   cmAnodeMainPnP2AxisZ.commandConfiguration.posRelative.direction := 0;
   cmAnodeMainPnP2AxisZ.commandConfiguration.posAbsolute.position := 3.0;
   cmAnodeMainPnP2AxisZ.commandConfiguration.posAbsolute.velocity := 30.0;
   cmAnodeMainPnP2AxisZ.commandConfiguration.posAbsolute.acceleration := 30.0;
   cmAnodeMainPnP2AxisZ.commandConfiguration.posAbsolute.deceleration := 30.0;
   cmAnodeMainPnP2AxisZ.commandConfiguration.posAbsolute.jerk := -1.0;
   cmAnodeMainPnP2AxisZ.commandConfiguration.posAbsolute.direction := 1;
   cmAnodeMainPnP2AxisZ.commandConfiguration.posAbsolute.positionChangeOnTheFly := FALSE;
   cmAnodeMainPnP2AxisZ.commandConfiguration.posAbsolute.velocityChangeOnTheFly := FALSE;
   cmAnodeMainPnP2AxisZ.commandConfiguration.posSuperimposed.distance := 0.0;
   cmAnodeMainPnP2AxisZ.commandConfiguration.posSuperimposed.velocityDiff := -1.0;
   cmAnodeMainPnP2AxisZ.commandConfiguration.posSuperimposed.acceleration := -1.0;
   cmAnodeMainPnP2AxisZ.commandConfiguration.posSuperimposed.deceleration := -1.0;
   cmAnodeMainPnP2AxisZ.commandConfiguration.posSuperimposed.jerk := -1.0;
   cmAnodeMainPnP2AxisZ.commandConfiguration.posSuperimposed.direction := 0;
   cmAnodeMainPnP2AxisZ.commandConfiguration.haltSuperimposed.deceleration := -1.0;
   cmAnodeMainPnP2AxisZ.commandConfiguration.haltSuperimposed.jerk := -1.0;
   cmAnodeMainPnP2AxisZ.commandConfiguration.haltSuperimposed.abortAcceleration := FALSE;
   cmAnodeMainPnP2AxisZ.commandConfiguration.gearInRelative.ratioNumerator := 1;
   cmAnodeMainPnP2AxisZ.commandConfiguration.gearInRelative.ratioDenominator := 1;
   cmAnodeMainPnP2AxisZ.commandConfiguration.gearInRelative.acceleration := -1.0;
   cmAnodeMainPnP2AxisZ.commandConfiguration.gearInRelative.deceleration := -1.0;
   cmAnodeMainPnP2AxisZ.commandConfiguration.gearInRelative.jerk := -1.0;
   cmAnodeMainPnP2AxisZ.commandConfiguration.gearInRelative.ratioChangeOnTheFly := FALSE;
   cmAnodeMainPnP2AxisZ.commandConfiguration.gearInAbsolute.ratioNumerator := 1;
   cmAnodeMainPnP2AxisZ.commandConfiguration.gearInAbsolute.ratioDenominator := 1;
   cmAnodeMainPnP2AxisZ.commandConfiguration.gearInAbsolute.masterSyncPosition := 0.0;
   cmAnodeMainPnP2AxisZ.commandConfiguration.gearInAbsolute.slaveSyncPosition := 0.0;
   cmAnodeMainPnP2AxisZ.commandConfiguration.gearInAbsolute.syncProfileReference := 1;
   cmAnodeMainPnP2AxisZ.commandConfiguration.gearInAbsolute.masterStartDistance := 0.0;
   cmAnodeMainPnP2AxisZ.commandConfiguration.gearInAbsolute.velocity := -1.0;
   cmAnodeMainPnP2AxisZ.commandConfiguration.gearInAbsolute.acceleration := -1.0;
   cmAnodeMainPnP2AxisZ.commandConfiguration.gearInAbsolute.deceleration := -1.0;
   cmAnodeMainPnP2AxisZ.commandConfiguration.gearInAbsolute.jerk := -1.0;
   cmAnodeMainPnP2AxisZ.commandConfiguration.gearInAbsolute.syncDirection := 1;
   cmAnodeMainPnP2AxisZ.commandConfiguration.gearInAbsolute.ratioChangeOnTheFly := FALSE;
   cmAnodeMainPnP2AxisZ.commandConfiguration.gearInVelocity.continuousUpdate := FALSE;
   cmAnodeMainPnP2AxisZ.commandConfiguration.gearInVelocity.ratioNumerator := 1;
   cmAnodeMainPnP2AxisZ.commandConfiguration.gearInVelocity.ratioDenominator := 1;
   cmAnodeMainPnP2AxisZ.commandConfiguration.gearInVelocity.acceleration := -1.0;
   cmAnodeMainPnP2AxisZ.commandConfiguration.gearInVelocity.deceleration := -1.0;
   cmAnodeMainPnP2AxisZ.commandConfiguration.gearInVelocity.jerk := -1.0;
   cmAnodeMainPnP2AxisZ.commandConfiguration.gearInVelocity.positionControlled := FALSE;
   cmAnodeMainPnP2AxisZ.commandConfiguration.camIn.masterOffset := 0.0;
   cmAnodeMainPnP2AxisZ.commandConfiguration.camIn.slaveOffset := 0.0;
   cmAnodeMainPnP2AxisZ.commandConfiguration.camIn.masterScaling := 1.0;
   cmAnodeMainPnP2AxisZ.commandConfiguration.camIn.slaveScaling := 1.0;
   cmAnodeMainPnP2AxisZ.commandConfiguration.camIn.masterSyncPosition := 0.0;
   cmAnodeMainPnP2AxisZ.commandConfiguration.camIn.syncProfileReference := 1;
   cmAnodeMainPnP2AxisZ.commandConfiguration.camIn.masterStartDistance := 0.0;
   cmAnodeMainPnP2AxisZ.commandConfiguration.camIn.velocity := -1.0;
   cmAnodeMainPnP2AxisZ.commandConfiguration.camIn.acceleration := -1.0;
   cmAnodeMainPnP2AxisZ.commandConfiguration.camIn.deceleration := -1.0;
   cmAnodeMainPnP2AxisZ.commandConfiguration.camIn.jerk := -1.0;
   cmAnodeMainPnP2AxisZ.commandConfiguration.camIn.applicationMode := 0;
   cmAnodeMainPnP2AxisZ.commandConfiguration.camIn.syncDirection := 1;
   cmAnodeMainPnP2AxisZ.commandConfiguration.gearOutCamOut.slavePosition := 0.0;
   cmAnodeMainPnP2AxisZ.commandConfiguration.gearOutCamOut.syncProfileReference := 1;
   cmAnodeMainPnP2AxisZ.commandConfiguration.gearOutCamOut.masterStopDistance := 0.0;
   cmAnodeMainPnP2AxisZ.commandConfiguration.gearOutCamOut.deceleration := -1.0;
   cmAnodeMainPnP2AxisZ.commandConfiguration.gearOutCamOut.jerk := -1.0;
   cmAnodeMainPnP2AxisZ.commandConfiguration.gearOutCamOut.syncOutDirection := 3;
   cmAnodeMainPnP2AxisZ.commandConfiguration.gearOutCamOut.gearOutCamOutMode := -1;
   cmAnodeMainPnP2AxisZ.commandConfiguration.phasing.phaseShift := 0.0;
   cmAnodeMainPnP2AxisZ.commandConfiguration.phasing.velocity := -1.0;
   cmAnodeMainPnP2AxisZ.commandConfiguration.phasing.acceleration := -1.0;
   cmAnodeMainPnP2AxisZ.commandConfiguration.phasing.deceleration := -1.0;
   cmAnodeMainPnP2AxisZ.commandConfiguration.phasing.jerk := -1.0;
   cmAnodeMainPnP2AxisZ.commandConfiguration.phasing.profileReference := 0;
   cmAnodeMainPnP2AxisZ.commandConfiguration.phasing.phasingDistance := 0.0;
   cmAnodeMainPnP2AxisZ.commandConfiguration.phasing.startPosition := 0.0;
   cmAnodeMainPnP2AxisZ.commandConfiguration.phasing.direction := 3;
   cmAnodeMainPnP2AxisZ.commandConfiguration.phasing.phaseAbsolute := TRUE;
   cmAnodeMainPnP2AxisZ.commandConfiguration.phasing.phaseShiftChangeOnTheFly := FALSE;
   cmAnodeMainPnP2AxisZ.commandConfiguration.offset.offset := 0.0;
   cmAnodeMainPnP2AxisZ.commandConfiguration.offset.profileReference := 1;
   cmAnodeMainPnP2AxisZ.commandConfiguration.offset.offsetDistance := 0.0;
   cmAnodeMainPnP2AxisZ.commandConfiguration.offset.startPosition := 0.0;
   cmAnodeMainPnP2AxisZ.commandConfiguration.offset.direction := 3;
   cmAnodeMainPnP2AxisZ.commandConfiguration.offset.offsetAbsolute := TRUE;
   cmAnodeMainPnP2AxisZ.commandConfiguration.offset.offsetChangeOnTheFly := FALSE;
   cmAnodeMainPnP2AxisZ.commands.enableAxis := FALSE;
   cmAnodeMainPnP2AxisZ.commands.resetAxis := FALSE;
   cmAnodeMainPnP2AxisZ.commands.openBrake := FALSE;
   cmAnodeMainPnP2AxisZ.commands.jogForward := FALSE;
   cmAnodeMainPnP2AxisZ.commands.jogBackward := FALSE;
   cmAnodeMainPnP2AxisZ.commands.moveVelocity := FALSE;
   cmAnodeMainPnP2AxisZ.commands.stop := FALSE;
   cmAnodeMainPnP2AxisZ.commands.fastStop := FALSE;
   cmAnodeMainPnP2AxisZ.commands.torqueLimiting := FALSE;
   cmAnodeMainPnP2AxisZ.commands.homing := FALSE;
   cmAnodeMainPnP2AxisZ.commands.posRelative := FALSE;
   cmAnodeMainPnP2AxisZ.commands.posAbsolute := FALSE;
   cmAnodeMainPnP2AxisZ.commands.posSuperimposed := FALSE;
   cmAnodeMainPnP2AxisZ.commands.haltSuperimposed := FALSE;
   cmAnodeMainPnP2AxisZ.commands.selectSetPosition := -1;
   cmAnodeMainPnP2AxisZ.commands.reset := FALSE;
   cmAnodeMainPnP2AxisZ.monitoring.valid := FALSE;
   cmAnodeMainPnP2AxisZ.monitoring.busy := TRUE;
   cmAnodeMainPnP2AxisZ.monitoring.error := TRUE;
   cmAnodeMainPnP2AxisZ.monitoring.status := 16#8600;
   cmAnodeMainPnP2AxisZ.monitoring.subfunctionStatus := 16#8001;
   cmAnodeMainPnP2AxisZ.monitoring.axisEnabled := FALSE;
   cmAnodeMainPnP2AxisZ.monitoring.resetActive := FALSE;
   cmAnodeMainPnP2AxisZ.monitoring.inVelocity := FALSE;
   cmAnodeMainPnP2AxisZ.monitoring.inLimitation := FALSE;
   cmAnodeMainPnP2AxisZ.monitoring.inClamping := FALSE;
   cmAnodeMainPnP2AxisZ.monitoring.startSync := FALSE;
   cmAnodeMainPnP2AxisZ.monitoring.inSync := FALSE;
   cmAnodeMainPnP2AxisZ.monitoring.inSimulation := FALSE;
   cmAnodeMainPnP2AxisZ.monitoring.jogSelected := FALSE;
   cmAnodeMainPnP2AxisZ.monitoring.moveVelocitySelected := FALSE;
   cmAnodeMainPnP2AxisZ.monitoring.stopSelected := FALSE;
   cmAnodeMainPnP2AxisZ.monitoring.fastStopSelected := FALSE;
   cmAnodeMainPnP2AxisZ.monitoring.torqueLimitingSelected := FALSE;
   cmAnodeMainPnP2AxisZ.monitoring.homingSelected := FALSE;
   cmAnodeMainPnP2AxisZ.monitoring.posRelativeSelected := FALSE;
   cmAnodeMainPnP2AxisZ.monitoring.posAbsoluteSelected := FALSE;
   cmAnodeMainPnP2AxisZ.monitoring.posSuperimposedSelected := FALSE;
   cmAnodeMainPnP2AxisZ.monitoring.haltSuperimposedSelected := FALSE;
   cmAnodeMainPnP2AxisZ.monitoring.commandBusy := FALSE;
   cmAnodeMainPnP2AxisZ.monitoring.commandDone := FALSE;
   cmAnodeMainPnP2AxisZ.monitoring.commandAborted := FALSE;
   cmAnodeMainPnP2AxisZ.monitoring.homingCommandBusy := FALSE;
   cmAnodeMainPnP2AxisZ.monitoring.homingCommandDone := FALSE;
   cmAnodeMainPnP2AxisZ.monitoring.homingCommandAborted := FALSE;
   cmAnodeMainPnP2AxisZ.monitoring.superimposedBusy := FALSE;
   cmAnodeMainPnP2AxisZ.monitoring.superimposedDone := FALSE;
   cmAnodeMainPnP2AxisZ.monitoring.superimposedAborted := FALSE;
   cmAnodeMainPnP2AxisZ.monitoring.actualPosition := 3.014;
   cmAnodeMainPnP2AxisZ.monitoring.actualSpeed := -0.00158945719401042;
   cmAnodeMainPnP2AxisZ.monitoring.speedUnit := 1062;
   cmAnodeMainPnP2AxisZ.monitoring.positionUnit := 1013;
   cmAnodeMainPnP2AxisZ.monitoring.axisType := 1;
   cmAnodeMainPnP2AxisZ.monitoring.interlockGeneralOut := TRUE;
   cmAnodeMainPnP2AxisZ.monitoring.interlockJogForwardOut := TRUE;
   cmAnodeMainPnP2AxisZ.monitoring.interlockJogBackwardOut := TRUE;
   cmAnodeAlignTableAxisX.commandConfiguration.generalSettings.stopOnError := TRUE;
   cmAnodeAlignTableAxisX.commandConfiguration.generalSettings.resetWithRestart := FALSE;
   cmAnodeAlignTableAxisX.commandConfiguration.generalSettings.abortWaitingSyncCmd := TRUE;
   cmAnodeAlignTableAxisX.commandConfiguration.power.startMode := 1;
   cmAnodeAlignTableAxisX.commandConfiguration.power.stopMode := 0;
   cmAnodeAlignTableAxisX.commandConfiguration.power.syncMotionSimulation := FALSE;
   cmAnodeAlignTableAxisX.commandConfiguration.power.syncMotionSimulationExtendedMode := -1;
   cmAnodeAlignTableAxisX.commandConfiguration.jog.velocity := 0.0;
   cmAnodeAlignTableAxisX.commandConfiguration.jog.acceleration := -1.0;
   cmAnodeAlignTableAxisX.commandConfiguration.jog.deceleration := -1.0;
   cmAnodeAlignTableAxisX.commandConfiguration.jog.jerk := -1.0;
   cmAnodeAlignTableAxisX.commandConfiguration.jog.positionControlled := TRUE;
   cmAnodeAlignTableAxisX.commandConfiguration.jog.increment := 0.0;
   cmAnodeAlignTableAxisX.commandConfiguration.jog.mode := 0;
   cmAnodeAlignTableAxisX.commandConfiguration.moveVelocity.velocity := 0.0;
   cmAnodeAlignTableAxisX.commandConfiguration.moveVelocity.acceleration := -1.0;
   cmAnodeAlignTableAxisX.commandConfiguration.moveVelocity.deceleration := -1.0;
   cmAnodeAlignTableAxisX.commandConfiguration.moveVelocity.jerk := -1.0;
   cmAnodeAlignTableAxisX.commandConfiguration.moveVelocity.direction := 0;
   cmAnodeAlignTableAxisX.commandConfiguration.moveVelocity.positionControlled := TRUE;
   cmAnodeAlignTableAxisX.commandConfiguration.moveVelocity.velocityChangeOnTheFly := FALSE;
   cmAnodeAlignTableAxisX.commandConfiguration.stop.deceleration := -1.0;
   cmAnodeAlignTableAxisX.commandConfiguration.stop.jerk := -1.0;
   cmAnodeAlignTableAxisX.commandConfiguration.stop.abortAcceleration := FALSE;
   cmAnodeAlignTableAxisX.commandConfiguration.fastStop.deceleration := -1.0;
   cmAnodeAlignTableAxisX.commandConfiguration.fastStop.jerk := -1.0;
   cmAnodeAlignTableAxisX.commandConfiguration.fastStop.abortAcceleration := FALSE;
   cmAnodeAlignTableAxisX.commandConfiguration.fastStop.replaceStopPossible := FALSE;
   cmAnodeAlignTableAxisX.commandConfiguration.torqueLimiting.limit := -1.0;
   cmAnodeAlignTableAxisX.commandConfiguration.torqueLimiting.mode := 0;
   cmAnodeAlignTableAxisX.commandConfiguration.homing.position := 0.0;
   cmAnodeAlignTableAxisX.commandConfiguration.homing.mode := 0;
   cmAnodeAlignTableAxisX.commandConfiguration.homing.sensor := 0;
   cmAnodeAlignTableAxisX.commandConfiguration.homing.extendedMode := -1;
   cmAnodeAlignTableAxisX.commandConfiguration.homing.extendedModeTorqueLimit := 0.0;
   cmAnodeAlignTableAxisX.commandConfiguration.homing.extendedModeTargetPosition := 0.0;
   cmAnodeAlignTableAxisX.commandConfiguration.posRelative.distance := 0.0;
   cmAnodeAlignTableAxisX.commandConfiguration.posRelative.velocity := -1.0;
   cmAnodeAlignTableAxisX.commandConfiguration.posRelative.acceleration := -1.0;
   cmAnodeAlignTableAxisX.commandConfiguration.posRelative.deceleration := -1.0;
   cmAnodeAlignTableAxisX.commandConfiguration.posRelative.jerk := -1.0;
   cmAnodeAlignTableAxisX.commandConfiguration.posRelative.direction := 0;
   cmAnodeAlignTableAxisX.commandConfiguration.posAbsolute.position := 0.0;
   cmAnodeAlignTableAxisX.commandConfiguration.posAbsolute.velocity := -1.0;
   cmAnodeAlignTableAxisX.commandConfiguration.posAbsolute.acceleration := -1.0;
   cmAnodeAlignTableAxisX.commandConfiguration.posAbsolute.deceleration := -1.0;
   cmAnodeAlignTableAxisX.commandConfiguration.posAbsolute.jerk := -1.0;
   cmAnodeAlignTableAxisX.commandConfiguration.posAbsolute.direction := 1;
   cmAnodeAlignTableAxisX.commandConfiguration.posAbsolute.positionChangeOnTheFly := FALSE;
   cmAnodeAlignTableAxisX.commandConfiguration.posAbsolute.velocityChangeOnTheFly := FALSE;
   cmAnodeAlignTableAxisX.commandConfiguration.posSuperimposed.distance := 0.0;
   cmAnodeAlignTableAxisX.commandConfiguration.posSuperimposed.velocityDiff := -1.0;
   cmAnodeAlignTableAxisX.commandConfiguration.posSuperimposed.acceleration := -1.0;
   cmAnodeAlignTableAxisX.commandConfiguration.posSuperimposed.deceleration := -1.0;
   cmAnodeAlignTableAxisX.commandConfiguration.posSuperimposed.jerk := -1.0;
   cmAnodeAlignTableAxisX.commandConfiguration.posSuperimposed.direction := 0;
   cmAnodeAlignTableAxisX.commandConfiguration.haltSuperimposed.deceleration := -1.0;
   cmAnodeAlignTableAxisX.commandConfiguration.haltSuperimposed.jerk := -1.0;
   cmAnodeAlignTableAxisX.commandConfiguration.haltSuperimposed.abortAcceleration := FALSE;
   cmAnodeAlignTableAxisX.commandConfiguration.gearInRelative.ratioNumerator := 1;
   cmAnodeAlignTableAxisX.commandConfiguration.gearInRelative.ratioDenominator := 1;
   cmAnodeAlignTableAxisX.commandConfiguration.gearInRelative.acceleration := -1.0;
   cmAnodeAlignTableAxisX.commandConfiguration.gearInRelative.deceleration := -1.0;
   cmAnodeAlignTableAxisX.commandConfiguration.gearInRelative.jerk := -1.0;
   cmAnodeAlignTableAxisX.commandConfiguration.gearInRelative.ratioChangeOnTheFly := FALSE;
   cmAnodeAlignTableAxisX.commandConfiguration.gearInAbsolute.ratioNumerator := 1;
   cmAnodeAlignTableAxisX.commandConfiguration.gearInAbsolute.ratioDenominator := 1;
   cmAnodeAlignTableAxisX.commandConfiguration.gearInAbsolute.masterSyncPosition := 0.0;
   cmAnodeAlignTableAxisX.commandConfiguration.gearInAbsolute.slaveSyncPosition := 0.0;
   cmAnodeAlignTableAxisX.commandConfiguration.gearInAbsolute.syncProfileReference := 1;
   cmAnodeAlignTableAxisX.commandConfiguration.gearInAbsolute.masterStartDistance := 0.0;
   cmAnodeAlignTableAxisX.commandConfiguration.gearInAbsolute.velocity := -1.0;
   cmAnodeAlignTableAxisX.commandConfiguration.gearInAbsolute.acceleration := -1.0;
   cmAnodeAlignTableAxisX.commandConfiguration.gearInAbsolute.deceleration := -1.0;
   cmAnodeAlignTableAxisX.commandConfiguration.gearInAbsolute.jerk := -1.0;
   cmAnodeAlignTableAxisX.commandConfiguration.gearInAbsolute.syncDirection := 1;
   cmAnodeAlignTableAxisX.commandConfiguration.gearInAbsolute.ratioChangeOnTheFly := FALSE;
   cmAnodeAlignTableAxisX.commandConfiguration.gearInVelocity.continuousUpdate := FALSE;
   cmAnodeAlignTableAxisX.commandConfiguration.gearInVelocity.ratioNumerator := 1;
   cmAnodeAlignTableAxisX.commandConfiguration.gearInVelocity.ratioDenominator := 1;
   cmAnodeAlignTableAxisX.commandConfiguration.gearInVelocity.acceleration := -1.0;
   cmAnodeAlignTableAxisX.commandConfiguration.gearInVelocity.deceleration := -1.0;
   cmAnodeAlignTableAxisX.commandConfiguration.gearInVelocity.jerk := -1.0;
   cmAnodeAlignTableAxisX.commandConfiguration.gearInVelocity.positionControlled := FALSE;
   cmAnodeAlignTableAxisX.commandConfiguration.camIn.masterOffset := 0.0;
   cmAnodeAlignTableAxisX.commandConfiguration.camIn.slaveOffset := 0.0;
   cmAnodeAlignTableAxisX.commandConfiguration.camIn.masterScaling := 1.0;
   cmAnodeAlignTableAxisX.commandConfiguration.camIn.slaveScaling := 1.0;
   cmAnodeAlignTableAxisX.commandConfiguration.camIn.masterSyncPosition := 0.0;
   cmAnodeAlignTableAxisX.commandConfiguration.camIn.syncProfileReference := 1;
   cmAnodeAlignTableAxisX.commandConfiguration.camIn.masterStartDistance := 0.0;
   cmAnodeAlignTableAxisX.commandConfiguration.camIn.velocity := -1.0;
   cmAnodeAlignTableAxisX.commandConfiguration.camIn.acceleration := -1.0;
   cmAnodeAlignTableAxisX.commandConfiguration.camIn.deceleration := -1.0;
   cmAnodeAlignTableAxisX.commandConfiguration.camIn.jerk := -1.0;
   cmAnodeAlignTableAxisX.commandConfiguration.camIn.applicationMode := 0;
   cmAnodeAlignTableAxisX.commandConfiguration.camIn.syncDirection := 1;
   cmAnodeAlignTableAxisX.commandConfiguration.gearOutCamOut.slavePosition := 0.0;
   cmAnodeAlignTableAxisX.commandConfiguration.gearOutCamOut.syncProfileReference := 1;
   cmAnodeAlignTableAxisX.commandConfiguration.gearOutCamOut.masterStopDistance := 0.0;
   cmAnodeAlignTableAxisX.commandConfiguration.gearOutCamOut.deceleration := -1.0;
   cmAnodeAlignTableAxisX.commandConfiguration.gearOutCamOut.jerk := -1.0;
   cmAnodeAlignTableAxisX.commandConfiguration.gearOutCamOut.syncOutDirection := 3;
   cmAnodeAlignTableAxisX.commandConfiguration.gearOutCamOut.gearOutCamOutMode := -1;
   cmAnodeAlignTableAxisX.commandConfiguration.phasing.phaseShift := 0.0;
   cmAnodeAlignTableAxisX.commandConfiguration.phasing.velocity := -1.0;
   cmAnodeAlignTableAxisX.commandConfiguration.phasing.acceleration := -1.0;
   cmAnodeAlignTableAxisX.commandConfiguration.phasing.deceleration := -1.0;
   cmAnodeAlignTableAxisX.commandConfiguration.phasing.jerk := -1.0;
   cmAnodeAlignTableAxisX.commandConfiguration.phasing.profileReference := 0;
   cmAnodeAlignTableAxisX.commandConfiguration.phasing.phasingDistance := 0.0;
   cmAnodeAlignTableAxisX.commandConfiguration.phasing.startPosition := 0.0;
   cmAnodeAlignTableAxisX.commandConfiguration.phasing.direction := 3;
   cmAnodeAlignTableAxisX.commandConfiguration.phasing.phaseAbsolute := TRUE;
   cmAnodeAlignTableAxisX.commandConfiguration.phasing.phaseShiftChangeOnTheFly := FALSE;
   cmAnodeAlignTableAxisX.commandConfiguration.offset.offset := 0.0;
   cmAnodeAlignTableAxisX.commandConfiguration.offset.profileReference := 1;
   cmAnodeAlignTableAxisX.commandConfiguration.offset.offsetDistance := 0.0;
   cmAnodeAlignTableAxisX.commandConfiguration.offset.startPosition := 0.0;
   cmAnodeAlignTableAxisX.commandConfiguration.offset.direction := 3;
   cmAnodeAlignTableAxisX.commandConfiguration.offset.offsetAbsolute := TRUE;
   cmAnodeAlignTableAxisX.commandConfiguration.offset.offsetChangeOnTheFly := FALSE;
   cmAnodeAlignTableAxisY1.commandConfiguration.generalSettings.stopOnError := TRUE;
   cmAnodeAlignTableAxisY1.commandConfiguration.generalSettings.resetWithRestart := FALSE;
   cmAnodeAlignTableAxisY1.commandConfiguration.generalSettings.abortWaitingSyncCmd := TRUE;
   cmAnodeAlignTableAxisY1.commandConfiguration.power.startMode := 1;
   cmAnodeAlignTableAxisY1.commandConfiguration.power.stopMode := 0;
   cmAnodeAlignTableAxisY1.commandConfiguration.power.syncMotionSimulation := FALSE;
   cmAnodeAlignTableAxisY1.commandConfiguration.power.syncMotionSimulationExtendedMode := -1;
   cmAnodeAlignTableAxisY1.commandConfiguration.jog.velocity := 0.0;
   cmAnodeAlignTableAxisY1.commandConfiguration.jog.acceleration := -1.0;
   cmAnodeAlignTableAxisY1.commandConfiguration.jog.deceleration := -1.0;
   cmAnodeAlignTableAxisY1.commandConfiguration.jog.jerk := -1.0;
   cmAnodeAlignTableAxisY1.commandConfiguration.jog.positionControlled := TRUE;
   cmAnodeAlignTableAxisY1.commandConfiguration.jog.increment := 0.0;
   cmAnodeAlignTableAxisY1.commandConfiguration.jog.mode := 0;
   cmAnodeAlignTableAxisY1.commandConfiguration.moveVelocity.velocity := 0.0;
   cmAnodeAlignTableAxisY1.commandConfiguration.moveVelocity.acceleration := -1.0;
   cmAnodeAlignTableAxisY1.commandConfiguration.moveVelocity.deceleration := -1.0;
   cmAnodeAlignTableAxisY1.commandConfiguration.moveVelocity.jerk := -1.0;
   cmAnodeAlignTableAxisY1.commandConfiguration.moveVelocity.direction := 0;
   cmAnodeAlignTableAxisY1.commandConfiguration.moveVelocity.positionControlled := TRUE;
   cmAnodeAlignTableAxisY1.commandConfiguration.moveVelocity.velocityChangeOnTheFly := FALSE;
   cmAnodeAlignTableAxisY1.commandConfiguration.stop.deceleration := -1.0;
   cmAnodeAlignTableAxisY1.commandConfiguration.stop.jerk := -1.0;
   cmAnodeAlignTableAxisY1.commandConfiguration.stop.abortAcceleration := FALSE;
   cmAnodeAlignTableAxisY1.commandConfiguration.fastStop.deceleration := -1.0;
   cmAnodeAlignTableAxisY1.commandConfiguration.fastStop.jerk := -1.0;
   cmAnodeAlignTableAxisY1.commandConfiguration.fastStop.abortAcceleration := FALSE;
   cmAnodeAlignTableAxisY1.commandConfiguration.fastStop.replaceStopPossible := FALSE;
   cmAnodeAlignTableAxisY1.commandConfiguration.torqueLimiting.limit := -1.0;
   cmAnodeAlignTableAxisY1.commandConfiguration.torqueLimiting.mode := 0;
   cmAnodeAlignTableAxisY1.commandConfiguration.homing.position := 0.0;
   cmAnodeAlignTableAxisY1.commandConfiguration.homing.mode := 0;
   cmAnodeAlignTableAxisY1.commandConfiguration.homing.sensor := 0;
   cmAnodeAlignTableAxisY1.commandConfiguration.homing.extendedMode := -1;
   cmAnodeAlignTableAxisY1.commandConfiguration.homing.extendedModeTorqueLimit := 0.0;
   cmAnodeAlignTableAxisY1.commandConfiguration.homing.extendedModeTargetPosition := 0.0;
   cmAnodeAlignTableAxisY1.commandConfiguration.posRelative.distance := 0.0;
   cmAnodeAlignTableAxisY1.commandConfiguration.posRelative.velocity := -1.0;
   cmAnodeAlignTableAxisY1.commandConfiguration.posRelative.acceleration := -1.0;
   cmAnodeAlignTableAxisY1.commandConfiguration.posRelative.deceleration := -1.0;
   cmAnodeAlignTableAxisY1.commandConfiguration.posRelative.jerk := -1.0;
   cmAnodeAlignTableAxisY1.commandConfiguration.posRelative.direction := 0;
   cmAnodeAlignTableAxisY1.commandConfiguration.posAbsolute.position := 0.0;
   cmAnodeAlignTableAxisY1.commandConfiguration.posAbsolute.velocity := -1.0;
   cmAnodeAlignTableAxisY1.commandConfiguration.posAbsolute.acceleration := -1.0;
   cmAnodeAlignTableAxisY1.commandConfiguration.posAbsolute.deceleration := -1.0;
   cmAnodeAlignTableAxisY1.commandConfiguration.posAbsolute.jerk := -1.0;
   cmAnodeAlignTableAxisY1.commandConfiguration.posAbsolute.direction := 1;
   cmAnodeAlignTableAxisY1.commandConfiguration.posAbsolute.positionChangeOnTheFly := FALSE;
   cmAnodeAlignTableAxisY1.commandConfiguration.posAbsolute.velocityChangeOnTheFly := FALSE;
   cmAnodeAlignTableAxisY1.commandConfiguration.posSuperimposed.distance := 0.0;
   cmAnodeAlignTableAxisY1.commandConfiguration.posSuperimposed.velocityDiff := -1.0;
   cmAnodeAlignTableAxisY1.commandConfiguration.posSuperimposed.acceleration := -1.0;
   cmAnodeAlignTableAxisY1.commandConfiguration.posSuperimposed.deceleration := -1.0;
   cmAnodeAlignTableAxisY1.commandConfiguration.posSuperimposed.jerk := -1.0;
   cmAnodeAlignTableAxisY1.commandConfiguration.posSuperimposed.direction := 0;
   cmAnodeAlignTableAxisY1.commandConfiguration.haltSuperimposed.deceleration := -1.0;
   cmAnodeAlignTableAxisY1.commandConfiguration.haltSuperimposed.jerk := -1.0;
   cmAnodeAlignTableAxisY1.commandConfiguration.haltSuperimposed.abortAcceleration := FALSE;
   cmAnodeAlignTableAxisY1.commandConfiguration.gearInRelative.ratioNumerator := 1;
   cmAnodeAlignTableAxisY1.commandConfiguration.gearInRelative.ratioDenominator := 1;
   cmAnodeAlignTableAxisY1.commandConfiguration.gearInRelative.acceleration := -1.0;
   cmAnodeAlignTableAxisY1.commandConfiguration.gearInRelative.deceleration := -1.0;
   cmAnodeAlignTableAxisY1.commandConfiguration.gearInRelative.jerk := -1.0;
   cmAnodeAlignTableAxisY1.commandConfiguration.gearInRelative.ratioChangeOnTheFly := FALSE;
   cmAnodeAlignTableAxisY1.commandConfiguration.gearInAbsolute.ratioNumerator := 1;
   cmAnodeAlignTableAxisY1.commandConfiguration.gearInAbsolute.ratioDenominator := 1;
   cmAnodeAlignTableAxisY1.commandConfiguration.gearInAbsolute.masterSyncPosition := 0.0;
   cmAnodeAlignTableAxisY1.commandConfiguration.gearInAbsolute.slaveSyncPosition := 0.0;
   cmAnodeAlignTableAxisY1.commandConfiguration.gearInAbsolute.syncProfileReference := 1;
   cmAnodeAlignTableAxisY1.commandConfiguration.gearInAbsolute.masterStartDistance := 0.0;
   cmAnodeAlignTableAxisY1.commandConfiguration.gearInAbsolute.velocity := -1.0;
   cmAnodeAlignTableAxisY1.commandConfiguration.gearInAbsolute.acceleration := -1.0;
   cmAnodeAlignTableAxisY1.commandConfiguration.gearInAbsolute.deceleration := -1.0;
   cmAnodeAlignTableAxisY1.commandConfiguration.gearInAbsolute.jerk := -1.0;
   cmAnodeAlignTableAxisY1.commandConfiguration.gearInAbsolute.syncDirection := 1;
   cmAnodeAlignTableAxisY1.commandConfiguration.gearInAbsolute.ratioChangeOnTheFly := FALSE;
   cmAnodeAlignTableAxisY1.commandConfiguration.gearInVelocity.continuousUpdate := FALSE;
   cmAnodeAlignTableAxisY1.commandConfiguration.gearInVelocity.ratioNumerator := 1;
   cmAnodeAlignTableAxisY1.commandConfiguration.gearInVelocity.ratioDenominator := 1;
   cmAnodeAlignTableAxisY1.commandConfiguration.gearInVelocity.acceleration := -1.0;
   cmAnodeAlignTableAxisY1.commandConfiguration.gearInVelocity.deceleration := -1.0;
   cmAnodeAlignTableAxisY1.commandConfiguration.gearInVelocity.jerk := -1.0;
   cmAnodeAlignTableAxisY1.commandConfiguration.gearInVelocity.positionControlled := FALSE;
   cmAnodeAlignTableAxisY1.commandConfiguration.camIn.masterOffset := 0.0;
   cmAnodeAlignTableAxisY1.commandConfiguration.camIn.slaveOffset := 0.0;
   cmAnodeAlignTableAxisY1.commandConfiguration.camIn.masterScaling := 1.0;
   cmAnodeAlignTableAxisY1.commandConfiguration.camIn.slaveScaling := 1.0;
   cmAnodeAlignTableAxisY1.commandConfiguration.camIn.masterSyncPosition := 0.0;
   cmAnodeAlignTableAxisY1.commandConfiguration.camIn.syncProfileReference := 1;
   cmAnodeAlignTableAxisY1.commandConfiguration.camIn.masterStartDistance := 0.0;
   cmAnodeAlignTableAxisY1.commandConfiguration.camIn.velocity := -1.0;
   cmAnodeAlignTableAxisY1.commandConfiguration.camIn.acceleration := -1.0;
   cmAnodeAlignTableAxisY1.commandConfiguration.camIn.deceleration := -1.0;
   cmAnodeAlignTableAxisY1.commandConfiguration.camIn.jerk := -1.0;
   cmAnodeAlignTableAxisY1.commandConfiguration.camIn.applicationMode := 0;
   cmAnodeAlignTableAxisY1.commandConfiguration.camIn.syncDirection := 1;
   cmAnodeAlignTableAxisY1.commandConfiguration.gearOutCamOut.slavePosition := 0.0;
   cmAnodeAlignTableAxisY1.commandConfiguration.gearOutCamOut.syncProfileReference := 1;
   cmAnodeAlignTableAxisY1.commandConfiguration.gearOutCamOut.masterStopDistance := 0.0;
   cmAnodeAlignTableAxisY1.commandConfiguration.gearOutCamOut.deceleration := -1.0;
   cmAnodeAlignTableAxisY1.commandConfiguration.gearOutCamOut.jerk := -1.0;
   cmAnodeAlignTableAxisY1.commandConfiguration.gearOutCamOut.syncOutDirection := 3;
   cmAnodeAlignTableAxisY1.commandConfiguration.gearOutCamOut.gearOutCamOutMode := -1;
   cmAnodeAlignTableAxisY1.commandConfiguration.phasing.phaseShift := 0.0;
   cmAnodeAlignTableAxisY1.commandConfiguration.phasing.velocity := -1.0;
   cmAnodeAlignTableAxisY1.commandConfiguration.phasing.acceleration := -1.0;
   cmAnodeAlignTableAxisY1.commandConfiguration.phasing.deceleration := -1.0;
   cmAnodeAlignTableAxisY1.commandConfiguration.phasing.jerk := -1.0;
   cmAnodeAlignTableAxisY1.commandConfiguration.phasing.profileReference := 0;
   cmAnodeAlignTableAxisY1.commandConfiguration.phasing.phasingDistance := 0.0;
   cmAnodeAlignTableAxisY1.commandConfiguration.phasing.startPosition := 0.0;
   cmAnodeAlignTableAxisY1.commandConfiguration.phasing.direction := 3;
   cmAnodeAlignTableAxisY1.commandConfiguration.phasing.phaseAbsolute := TRUE;
   cmAnodeAlignTableAxisY1.commandConfiguration.phasing.phaseShiftChangeOnTheFly := FALSE;
   cmAnodeAlignTableAxisY1.commandConfiguration.offset.offset := 0.0;
   cmAnodeAlignTableAxisY1.commandConfiguration.offset.profileReference := 1;
   cmAnodeAlignTableAxisY1.commandConfiguration.offset.offsetDistance := 0.0;
   cmAnodeAlignTableAxisY1.commandConfiguration.offset.startPosition := 0.0;
   cmAnodeAlignTableAxisY1.commandConfiguration.offset.direction := 3;
   cmAnodeAlignTableAxisY1.commandConfiguration.offset.offsetAbsolute := TRUE;
   cmAnodeAlignTableAxisY1.commandConfiguration.offset.offsetChangeOnTheFly := FALSE;
   cmAnodeAlignTableAxisY1.monitoring.valid := FALSE;
   cmAnodeAlignTableAxisY1.monitoring.busy := TRUE;
   cmAnodeAlignTableAxisY1.monitoring.error := TRUE;
   cmAnodeAlignTableAxisY1.monitoring.status := 16#8600;
   cmAnodeAlignTableAxisY1.monitoring.subfunctionStatus := 16#8001;
   cmAnodeAlignTableAxisY1.monitoring.axisEnabled := FALSE;
   cmAnodeAlignTableAxisY1.monitoring.resetActive := FALSE;
   cmAnodeAlignTableAxisY1.monitoring.inVelocity := FALSE;
   cmAnodeAlignTableAxisY1.monitoring.inLimitation := FALSE;
   cmAnodeAlignTableAxisY1.monitoring.inClamping := FALSE;
   cmAnodeAlignTableAxisY1.monitoring.startSync := FALSE;
   cmAnodeAlignTableAxisY1.monitoring.inSync := FALSE;
   cmAnodeAlignTableAxisY1.monitoring.inSimulation := FALSE;
   cmAnodeAlignTableAxisY1.monitoring.jogSelected := FALSE;
   cmAnodeAlignTableAxisY1.monitoring.moveVelocitySelected := FALSE;
   cmAnodeAlignTableAxisY1.monitoring.stopSelected := FALSE;
   cmAnodeAlignTableAxisY1.monitoring.fastStopSelected := FALSE;
   cmAnodeAlignTableAxisY1.monitoring.torqueLimitingSelected := FALSE;
   cmAnodeAlignTableAxisY1.monitoring.homingSelected := FALSE;
   cmAnodeAlignTableAxisY1.monitoring.posRelativeSelected := FALSE;
   cmAnodeAlignTableAxisY1.monitoring.posAbsoluteSelected := FALSE;
   cmAnodeAlignTableAxisY1.monitoring.posSuperimposedSelected := FALSE;
   cmAnodeAlignTableAxisY1.monitoring.haltSuperimposedSelected := FALSE;
   cmAnodeAlignTableAxisY1.monitoring.commandBusy := FALSE;
   cmAnodeAlignTableAxisY1.monitoring.commandDone := FALSE;
   cmAnodeAlignTableAxisY1.monitoring.commandAborted := FALSE;
   cmAnodeAlignTableAxisY1.monitoring.homingCommandBusy := FALSE;
   cmAnodeAlignTableAxisY1.monitoring.homingCommandDone := FALSE;
   cmAnodeAlignTableAxisY1.monitoring.homingCommandAborted := FALSE;
   cmAnodeAlignTableAxisY1.monitoring.superimposedBusy := FALSE;
   cmAnodeAlignTableAxisY1.monitoring.superimposedDone := FALSE;
   cmAnodeAlignTableAxisY1.monitoring.superimposedAborted := FALSE;
   cmAnodeAlignTableAxisY1.monitoring.actualPosition := 0.6;
   cmAnodeAlignTableAxisY1.monitoring.actualSpeed := 0.0;
   cmAnodeAlignTableAxisY1.monitoring.speedUnit := 1062;
   cmAnodeAlignTableAxisY1.monitoring.positionUnit := 1013;
   cmAnodeAlignTableAxisY1.monitoring.axisType := 1;
   cmAnodeAlignTableAxisY1.monitoring.interlockGeneralOut := TRUE;
   cmAnodeAlignTableAxisY1.monitoring.interlockJogForwardOut := TRUE;
   cmAnodeAlignTableAxisY1.monitoring.interlockJogBackwardOut := TRUE;
   cmAnodeAlignTableAxisY2.commandConfiguration.generalSettings.stopOnError := TRUE;
   cmAnodeAlignTableAxisY2.commandConfiguration.generalSettings.resetWithRestart := FALSE;
   cmAnodeAlignTableAxisY2.commandConfiguration.generalSettings.abortWaitingSyncCmd := TRUE;
   cmAnodeAlignTableAxisY2.commandConfiguration.power.startMode := 1;
   cmAnodeAlignTableAxisY2.commandConfiguration.power.stopMode := 0;
   cmAnodeAlignTableAxisY2.commandConfiguration.power.syncMotionSimulation := FALSE;
   cmAnodeAlignTableAxisY2.commandConfiguration.power.syncMotionSimulationExtendedMode := -1;
   cmAnodeAlignTableAxisY2.commandConfiguration.jog.velocity := 0.0;
   cmAnodeAlignTableAxisY2.commandConfiguration.jog.acceleration := -1.0;
   cmAnodeAlignTableAxisY2.commandConfiguration.jog.deceleration := -1.0;
   cmAnodeAlignTableAxisY2.commandConfiguration.jog.jerk := -1.0;
   cmAnodeAlignTableAxisY2.commandConfiguration.jog.positionControlled := TRUE;
   cmAnodeAlignTableAxisY2.commandConfiguration.jog.increment := 0.0;
   cmAnodeAlignTableAxisY2.commandConfiguration.jog.mode := 0;
   cmAnodeAlignTableAxisY2.commandConfiguration.moveVelocity.velocity := 0.0;
   cmAnodeAlignTableAxisY2.commandConfiguration.moveVelocity.acceleration := -1.0;
   cmAnodeAlignTableAxisY2.commandConfiguration.moveVelocity.deceleration := -1.0;
   cmAnodeAlignTableAxisY2.commandConfiguration.moveVelocity.jerk := -1.0;
   cmAnodeAlignTableAxisY2.commandConfiguration.moveVelocity.direction := 0;
   cmAnodeAlignTableAxisY2.commandConfiguration.moveVelocity.positionControlled := TRUE;
   cmAnodeAlignTableAxisY2.commandConfiguration.moveVelocity.velocityChangeOnTheFly := FALSE;
   cmAnodeAlignTableAxisY2.commandConfiguration.stop.deceleration := -1.0;
   cmAnodeAlignTableAxisY2.commandConfiguration.stop.jerk := -1.0;
   cmAnodeAlignTableAxisY2.commandConfiguration.stop.abortAcceleration := FALSE;
   cmAnodeAlignTableAxisY2.commandConfiguration.fastStop.deceleration := -1.0;
   cmAnodeAlignTableAxisY2.commandConfiguration.fastStop.jerk := -1.0;
   cmAnodeAlignTableAxisY2.commandConfiguration.fastStop.abortAcceleration := FALSE;
   cmAnodeAlignTableAxisY2.commandConfiguration.fastStop.replaceStopPossible := FALSE;
   cmAnodeAlignTableAxisY2.commandConfiguration.torqueLimiting.limit := -1.0;
   cmAnodeAlignTableAxisY2.commandConfiguration.torqueLimiting.mode := 0;
   cmAnodeAlignTableAxisY2.commandConfiguration.homing.position := 0.0;
   cmAnodeAlignTableAxisY2.commandConfiguration.homing.mode := 0;
   cmAnodeAlignTableAxisY2.commandConfiguration.homing.sensor := 0;
   cmAnodeAlignTableAxisY2.commandConfiguration.homing.extendedMode := -1;
   cmAnodeAlignTableAxisY2.commandConfiguration.homing.extendedModeTorqueLimit := 0.0;
   cmAnodeAlignTableAxisY2.commandConfiguration.homing.extendedModeTargetPosition := 0.0;
   cmAnodeAlignTableAxisY2.commandConfiguration.posRelative.distance := 0.0;
   cmAnodeAlignTableAxisY2.commandConfiguration.posRelative.velocity := -1.0;
   cmAnodeAlignTableAxisY2.commandConfiguration.posRelative.acceleration := -1.0;
   cmAnodeAlignTableAxisY2.commandConfiguration.posRelative.deceleration := -1.0;
   cmAnodeAlignTableAxisY2.commandConfiguration.posRelative.jerk := -1.0;
   cmAnodeAlignTableAxisY2.commandConfiguration.posRelative.direction := 0;
   cmAnodeAlignTableAxisY2.commandConfiguration.posAbsolute.position := 0.0;
   cmAnodeAlignTableAxisY2.commandConfiguration.posAbsolute.velocity := -1.0;
   cmAnodeAlignTableAxisY2.commandConfiguration.posAbsolute.acceleration := -1.0;
   cmAnodeAlignTableAxisY2.commandConfiguration.posAbsolute.deceleration := -1.0;
   cmAnodeAlignTableAxisY2.commandConfiguration.posAbsolute.jerk := -1.0;
   cmAnodeAlignTableAxisY2.commandConfiguration.posAbsolute.direction := 1;
   cmAnodeAlignTableAxisY2.commandConfiguration.posAbsolute.positionChangeOnTheFly := FALSE;
   cmAnodeAlignTableAxisY2.commandConfiguration.posAbsolute.velocityChangeOnTheFly := FALSE;
   cmAnodeAlignTableAxisY2.commandConfiguration.posSuperimposed.distance := 0.0;
   cmAnodeAlignTableAxisY2.commandConfiguration.posSuperimposed.velocityDiff := -1.0;
   cmAnodeAlignTableAxisY2.commandConfiguration.posSuperimposed.acceleration := -1.0;
   cmAnodeAlignTableAxisY2.commandConfiguration.posSuperimposed.deceleration := -1.0;
   cmAnodeAlignTableAxisY2.commandConfiguration.posSuperimposed.jerk := -1.0;
   cmAnodeAlignTableAxisY2.commandConfiguration.posSuperimposed.direction := 0;
   cmAnodeAlignTableAxisY2.commandConfiguration.haltSuperimposed.deceleration := -1.0;
   cmAnodeAlignTableAxisY2.commandConfiguration.haltSuperimposed.jerk := -1.0;
   cmAnodeAlignTableAxisY2.commandConfiguration.haltSuperimposed.abortAcceleration := FALSE;
   cmAnodeAlignTableAxisY2.commandConfiguration.gearInRelative.ratioNumerator := 1;
   cmAnodeAlignTableAxisY2.commandConfiguration.gearInRelative.ratioDenominator := 1;
   cmAnodeAlignTableAxisY2.commandConfiguration.gearInRelative.acceleration := -1.0;
   cmAnodeAlignTableAxisY2.commandConfiguration.gearInRelative.deceleration := -1.0;
   cmAnodeAlignTableAxisY2.commandConfiguration.gearInRelative.jerk := -1.0;
   cmAnodeAlignTableAxisY2.commandConfiguration.gearInRelative.ratioChangeOnTheFly := FALSE;
   cmAnodeAlignTableAxisY2.commandConfiguration.gearInAbsolute.ratioNumerator := 1;
   cmAnodeAlignTableAxisY2.commandConfiguration.gearInAbsolute.ratioDenominator := 1;
   cmAnodeAlignTableAxisY2.commandConfiguration.gearInAbsolute.masterSyncPosition := 0.0;
   cmAnodeAlignTableAxisY2.commandConfiguration.gearInAbsolute.slaveSyncPosition := 0.0;
   cmAnodeAlignTableAxisY2.commandConfiguration.gearInAbsolute.syncProfileReference := 1;
   cmAnodeAlignTableAxisY2.commandConfiguration.gearInAbsolute.masterStartDistance := 0.0;
   cmAnodeAlignTableAxisY2.commandConfiguration.gearInAbsolute.velocity := -1.0;
   cmAnodeAlignTableAxisY2.commandConfiguration.gearInAbsolute.acceleration := -1.0;
   cmAnodeAlignTableAxisY2.commandConfiguration.gearInAbsolute.deceleration := -1.0;
   cmAnodeAlignTableAxisY2.commandConfiguration.gearInAbsolute.jerk := -1.0;
   cmAnodeAlignTableAxisY2.commandConfiguration.gearInAbsolute.syncDirection := 1;
   cmAnodeAlignTableAxisY2.commandConfiguration.gearInAbsolute.ratioChangeOnTheFly := FALSE;
   cmAnodeAlignTableAxisY2.commandConfiguration.gearInVelocity.continuousUpdate := FALSE;
   cmAnodeAlignTableAxisY2.commandConfiguration.gearInVelocity.ratioNumerator := 1;
   cmAnodeAlignTableAxisY2.commandConfiguration.gearInVelocity.ratioDenominator := 1;
   cmAnodeAlignTableAxisY2.commandConfiguration.gearInVelocity.acceleration := -1.0;
   cmAnodeAlignTableAxisY2.commandConfiguration.gearInVelocity.deceleration := -1.0;
   cmAnodeAlignTableAxisY2.commandConfiguration.gearInVelocity.jerk := -1.0;
   cmAnodeAlignTableAxisY2.commandConfiguration.gearInVelocity.positionControlled := FALSE;
   cmAnodeAlignTableAxisY2.commandConfiguration.camIn.masterOffset := 0.0;
   cmAnodeAlignTableAxisY2.commandConfiguration.camIn.slaveOffset := 0.0;
   cmAnodeAlignTableAxisY2.commandConfiguration.camIn.masterScaling := 1.0;
   cmAnodeAlignTableAxisY2.commandConfiguration.camIn.slaveScaling := 1.0;
   cmAnodeAlignTableAxisY2.commandConfiguration.camIn.masterSyncPosition := 0.0;
   cmAnodeAlignTableAxisY2.commandConfiguration.camIn.syncProfileReference := 1;
   cmAnodeAlignTableAxisY2.commandConfiguration.camIn.masterStartDistance := 0.0;
   cmAnodeAlignTableAxisY2.commandConfiguration.camIn.velocity := -1.0;
   cmAnodeAlignTableAxisY2.commandConfiguration.camIn.acceleration := -1.0;
   cmAnodeAlignTableAxisY2.commandConfiguration.camIn.deceleration := -1.0;
   cmAnodeAlignTableAxisY2.commandConfiguration.camIn.jerk := -1.0;
   cmAnodeAlignTableAxisY2.commandConfiguration.camIn.applicationMode := 0;
   cmAnodeAlignTableAxisY2.commandConfiguration.camIn.syncDirection := 1;
   cmAnodeAlignTableAxisY2.commandConfiguration.gearOutCamOut.slavePosition := 0.0;
   cmAnodeAlignTableAxisY2.commandConfiguration.gearOutCamOut.syncProfileReference := 1;
   cmAnodeAlignTableAxisY2.commandConfiguration.gearOutCamOut.masterStopDistance := 0.0;
   cmAnodeAlignTableAxisY2.commandConfiguration.gearOutCamOut.deceleration := -1.0;
   cmAnodeAlignTableAxisY2.commandConfiguration.gearOutCamOut.jerk := -1.0;
   cmAnodeAlignTableAxisY2.commandConfiguration.gearOutCamOut.syncOutDirection := 3;
   cmAnodeAlignTableAxisY2.commandConfiguration.gearOutCamOut.gearOutCamOutMode := -1;
   cmAnodeAlignTableAxisY2.commandConfiguration.phasing.phaseShift := 0.0;
   cmAnodeAlignTableAxisY2.commandConfiguration.phasing.velocity := -1.0;
   cmAnodeAlignTableAxisY2.commandConfiguration.phasing.acceleration := -1.0;
   cmAnodeAlignTableAxisY2.commandConfiguration.phasing.deceleration := -1.0;
   cmAnodeAlignTableAxisY2.commandConfiguration.phasing.jerk := -1.0;
   cmAnodeAlignTableAxisY2.commandConfiguration.phasing.profileReference := 0;
   cmAnodeAlignTableAxisY2.commandConfiguration.phasing.phasingDistance := 0.0;
   cmAnodeAlignTableAxisY2.commandConfiguration.phasing.startPosition := 0.0;
   cmAnodeAlignTableAxisY2.commandConfiguration.phasing.direction := 3;
   cmAnodeAlignTableAxisY2.commandConfiguration.phasing.phaseAbsolute := TRUE;
   cmAnodeAlignTableAxisY2.commandConfiguration.phasing.phaseShiftChangeOnTheFly := FALSE;
   cmAnodeAlignTableAxisY2.commandConfiguration.offset.offset := 0.0;
   cmAnodeAlignTableAxisY2.commandConfiguration.offset.profileReference := 1;
   cmAnodeAlignTableAxisY2.commandConfiguration.offset.offsetDistance := 0.0;
   cmAnodeAlignTableAxisY2.commandConfiguration.offset.startPosition := 0.0;
   cmAnodeAlignTableAxisY2.commandConfiguration.offset.direction := 3;
   cmAnodeAlignTableAxisY2.commandConfiguration.offset.offsetAbsolute := TRUE;
   cmAnodeAlignTableAxisY2.commandConfiguration.offset.offsetChangeOnTheFly := FALSE;
   cmAnodeAlignTableAxisY2.monitoring.valid := FALSE;
   cmAnodeAlignTableAxisY2.monitoring.busy := TRUE;
   cmAnodeAlignTableAxisY2.monitoring.error := TRUE;
   cmAnodeAlignTableAxisY2.monitoring.status := 16#8600;
   cmAnodeAlignTableAxisY2.monitoring.subfunctionStatus := 16#8001;
   cmAnodeAlignTableAxisY2.monitoring.axisEnabled := FALSE;
   cmAnodeAlignTableAxisY2.monitoring.resetActive := FALSE;
   cmAnodeAlignTableAxisY2.monitoring.inVelocity := FALSE;
   cmAnodeAlignTableAxisY2.monitoring.inLimitation := FALSE;
   cmAnodeAlignTableAxisY2.monitoring.inClamping := FALSE;
   cmAnodeAlignTableAxisY2.monitoring.startSync := FALSE;
   cmAnodeAlignTableAxisY2.monitoring.inSync := FALSE;
   cmAnodeAlignTableAxisY2.monitoring.inSimulation := FALSE;
   cmAnodeAlignTableAxisY2.monitoring.jogSelected := FALSE;
   cmAnodeAlignTableAxisY2.monitoring.moveVelocitySelected := FALSE;
   cmAnodeAlignTableAxisY2.monitoring.stopSelected := FALSE;
   cmAnodeAlignTableAxisY2.monitoring.fastStopSelected := FALSE;
   cmAnodeAlignTableAxisY2.monitoring.torqueLimitingSelected := FALSE;
   cmAnodeAlignTableAxisY2.monitoring.homingSelected := FALSE;
   cmAnodeAlignTableAxisY2.monitoring.posRelativeSelected := FALSE;
   cmAnodeAlignTableAxisY2.monitoring.posAbsoluteSelected := FALSE;
   cmAnodeAlignTableAxisY2.monitoring.posSuperimposedSelected := FALSE;
   cmAnodeAlignTableAxisY2.monitoring.haltSuperimposedSelected := FALSE;
   cmAnodeAlignTableAxisY2.monitoring.commandBusy := FALSE;
   cmAnodeAlignTableAxisY2.monitoring.commandDone := FALSE;
   cmAnodeAlignTableAxisY2.monitoring.commandAborted := FALSE;
   cmAnodeAlignTableAxisY2.monitoring.homingCommandBusy := FALSE;
   cmAnodeAlignTableAxisY2.monitoring.homingCommandDone := FALSE;
   cmAnodeAlignTableAxisY2.monitoring.homingCommandAborted := FALSE;
   cmAnodeAlignTableAxisY2.monitoring.superimposedBusy := FALSE;
   cmAnodeAlignTableAxisY2.monitoring.superimposedDone := FALSE;
   cmAnodeAlignTableAxisY2.monitoring.superimposedAborted := FALSE;
   cmAnodeAlignTableAxisY2.monitoring.actualPosition := 0.0;
   cmAnodeAlignTableAxisY2.monitoring.actualSpeed := 0.0;
   cmAnodeAlignTableAxisY2.monitoring.speedUnit := 1062;
   cmAnodeAlignTableAxisY2.monitoring.positionUnit := 1013;
   cmAnodeAlignTableAxisY2.monitoring.axisType := 1;
   cmAnodeAlignTableAxisY2.monitoring.interlockGeneralOut := TRUE;
   cmAnodeAlignTableAxisY2.monitoring.interlockJogForwardOut := TRUE;
   cmAnodeAlignTableAxisY2.monitoring.interlockJogBackwardOut := TRUE;
   cmAnodeMainPnP1RotaryCwCcw.commands.commandHomePos := FALSE;
   cmAnodeMainPnP1RotaryCwCcw.commands.commandWorkPos := FALSE;
   cmAnodeMainPnP1RotaryCwCcw.commands.reset := FALSE;
   cmAnodeMainPnP1RotaryCwCcw.monitoring.valid := TRUE;
   cmAnodeMainPnP1RotaryCwCcw.monitoring.busy := TRUE;
   cmAnodeMainPnP1RotaryCwCcw.monitoring.error := FALSE;
   cmAnodeMainPnP1RotaryCwCcw.monitoring.status := 16#7100;
   cmAnodeMainPnP1RotaryCwCcw.monitoring.inHomePos := FALSE;
   cmAnodeMainPnP1RotaryCwCcw.monitoring.inWorkPos := FALSE;
   cmAnodeMainPnP1RotaryCwCcw.monitoring.interlockWorkPosOut := FALSE;
   cmAnodeMainPnP1RotaryCwCcw.monitoring.interlockHomePosOut := FALSE;
   cmAnodeMainPnP1SuctionPlateVacuum.commands.commandHomePos := FALSE;
   cmAnodeMainPnP1SuctionPlateVacuum.commands.commandWorkPos := FALSE;
   cmAnodeMainPnP1SuctionPlateVacuum.commands.reset := FALSE;
   cmAnodeMainPnP2SuctionPlateVacuum.commands.commandHomePos := FALSE;
   cmAnodeMainPnP2SuctionPlateVacuum.commands.commandWorkPos := FALSE;
   cmAnodeMainPnP2SuctionPlateVacuum.commands.reset := FALSE;
   cmAnodeAlignTableSuctionPlateVacuum.commands.commandHomePos := FALSE;
   cmAnodeAlignTableSuctionPlateVacuum.commands.commandWorkPos := FALSE;
   cmAnodeAlignTableSuctionPlateVacuum.commands.reset := FALSE;
   cmAnodeNgBoxLockUpDown.commands.commandHomePos := FALSE;
   cmAnodeNgBoxLockUpDown.commands.commandWorkPos := FALSE;
   cmAnodeNgBoxLockUpDown.commands.reset := FALSE;
   cmAnodeNgBoxLockUpDown.monitoring.valid := TRUE;
   cmAnodeNgBoxLockUpDown.monitoring.busy := TRUE;
   cmAnodeNgBoxLockUpDown.monitoring.error := FALSE;
   cmAnodeNgBoxLockUpDown.monitoring.status := 16#7003;
   cmAnodeNgBoxLockUpDown.monitoring.inHomePos := TRUE;
   cmAnodeNgBoxLockUpDown.monitoring.inWorkPos := FALSE;
   cmAnodeNgBoxLockUpDown.monitoring.interlockWorkPosOut := TRUE;
   cmAnodeNgBoxLockUpDown.monitoring.interlockHomePosOut := TRUE;
END_DATA_BLOCK
